TYPE TupleStruct__2:
    STRUCT
        field1: DINT;
        field2: DINT;
    END_STRUCT
END_TYPE

(* stored: ProductVersion 3.1.0.18, Version 1.1.0.1 *)
